// TwinCAT 3 PLC project TcOtel_Tester
// ProgramVersion: 3.1.4026.22
// CompilerDefines: DEBUG
// libraries:
//   TcOtel, * (AVM Engineering)
//   Tc2_Standard, * (Beckhoff Automation GmbH)
//   Tc2_System, * (Beckhoff Automation GmbH)
//   Tc2_Utilities, * (Beckhoff Automation GmbH)
//   Tc3_Module, * (Beckhoff Automation GmbH)
//   Base Interfaces,newest,System
// project tree:
//   GVLs/ GVL.TcGVL, GVL_TracePropagation.TcGVL
//   / PlcTask.TcTTO
//   POUs/ CheckBounds.TcPOU, CheckLRangeSigned.TcPOU, CheckLRangeUnsigned.TcPOU, CheckPointer.TcPOU, CheckRangeSigned.TcPOU, CheckRangeUnsigned.TcPOU, FB_Motor.TcPOU (not stored), FB_TcExternalTime.TcPOU, F_FUN.TcPOU (excluded from build), MAIN.TcPOU (not stored), PRG_TestMetricApi.TcPOU, PRG_TestSimpleApi.TcPOU (not stored), PRG_TestTraceApi.TcPOU, PRG_TestTracePropagation.TcPOU, PRG_TestTracerInstance.TcPOU
// (motion and I/O tree: see PLC project tcotel)
// real-time tasks:
//   TASK PlcTask: cycle T#1ms, priority 20, ADS port 350

CONFIGURATION TcOtel_Tester
    RESOURCE PLC ON TwinCAT3
        TASK PlcTask(INTERVAL := T#1ms, PRIORITY := 20);
        PROGRAM MAIN WITH PlcTask : MAIN;
    END_RESOURCE
END_CONFIGURATION

// ---- GVLs/GVL.TcGVL
{attribute 'qualified_only'}
VAR_GLOBAL
END_VAR

// ---- GVLs/GVL_TracePropagation.TcGVL
(*
Shared state for the Phase-5 cross-task propagation live test
(PRG_TestTracePropagation). Kept in a GVL so one PRG can produce a
traceparent string and another — or a later scenario in the same PRG
— can consume it across cycles.
*)
{attribute 'qualified_only'}
VAR_GLOBAL
    (* Pattern A: explicit W3C traceparent handed off between producer
       and consumer. 55 chars is enough for 00-<32hex>-<16hex>-01. *)
    sCurrentTraceParent : STRING(60);

    (* Pattern D: workpiece-centric trace_id derived via hash of the
       physical workpiece identifier. Modules that can see the ID but
       not a data bus can still aggregate their spans under one
       trace_id. *)
    sWorkpieceId        : STRING(40);
END_VAR

// ---- POUs/PRG_TestTracePropagation.TcPOU
(*
:Description: Phase-5 live cross-task propagation scenarios.

Runs three scenarios on a round-robin cadence so tc-otel sees all
three patterns documented in docs/traces-propagation.md:

  Scenario 1 (Pattern A — explicit traceparent handoff):
    Producer opens a Client span 'order_submit', reads its own
    TraceParent property before End, parks the string in the GVL.
    Consumer later opens 'handle_order' via the FB_Span.Begin
    overload with sTraceParent := the parked string. Tempo should
    render a two-span tree (Client → Server).

  Scenario 2 (Pattern D — workpiece-centric hash):
    Synthesises a workpiece_id like "WP-1234", builds a W3C header
    via F_TraceParentFromString (all-zero span_id — no upstream
    station cited). Opens three module spans across three cycles,
    each passing the same header. Tempo should show one trace with
    three sibling spans sharing a trace_id.

  Scenario 3 (chained producer-consumer-consumer):
    Each stage reads its own TraceParent property before End(),
    passes it to the next stage's Begin. Uses per-instance access
    so parallel Scenarios 1 and 2 on the same task can't poison
    the task-global CurrentTraceParent stack. Tempo shows a linear
    chain A → B → C.

All scenarios use FB_Span methods only — no low-level tracer access.
*)
PROGRAM PRG_TestTracePropagation
VAR
    tracer         : FB_Trace;

    (* Scenario 1: explicit handoff *)
    spnProducer    : FB_Span(tracer);
    spnConsumer    : FB_Span(tracer);
    tScenario1Acc  : TIME;
    nScenario1Step : USINT;  (* 0 idle, 1 producer open, 2 producer ended, 3 consumer open *)

    (* Scenario 2: hash-based, no handoff *)
    spnStageA      : FB_Span(tracer);
    spnStageB      : FB_Span(tracer);
    spnStageC      : FB_Span(tracer);
    tScenario2Acc  : TIME;
    nScenario2Step : USINT;  (* 0..3 *)
    nWorkpieceSeq  : DINT;
    sTraceParentHash : STRING(60);

    (* Scenario 3: chained *)
    spnChainA      : FB_Span(tracer);
    spnChainB      : FB_Span(tracer);
    spnChainC      : FB_Span(tracer);
    tScenario3Acc  : TIME;
    nScenario3Step : USINT;
    sChainTp1      : STRING(60);
    sChainTp2      : STRING(60);

    nSeq           : DINT;
END_VAR


// ─── Scenario 1: explicit traceparent handoff (every 3 s) ───
tScenario1Acc := tScenario1Acc + T#1MS;

CASE nScenario1Step OF
0:  // idle — wait for 3 s cycle start
    IF tScenario1Acc >= T#3S THEN
        tScenario1Acc := T#0S;
        spnProducer.Begin('order_submit', eKind := E_SpanKind.eClient);
        spnProducer.AddInt('seq', nSeq);
        nScenario1Step := 1;
    END_IF
1:  // producer open for ~100 ms, then capture traceparent + end
    IF tScenario1Acc >= T#100MS THEN
        GVL_TracePropagation.sCurrentTraceParent := spnProducer.TraceParent;
        spnProducer.AddEvent('traceparent_captured');
        spnProducer.End();
        nScenario1Step := 2;
    END_IF
2:  // 50 ms gap between producer End and consumer Begin — exercises
    // the "producer already flushed, consumer still opens as child"
    // code path in tc-otel.
    IF tScenario1Acc >= T#150MS THEN
        spnConsumer.Begin(
            sName        := 'handle_order',
            eKind        := E_SpanKind.eServer,
            sTraceParent := GVL_TracePropagation.sCurrentTraceParent);
        spnConsumer.AddInt('seq', nSeq);
		F_Log(E_LogLevel.eDebug, 'Try add trace reference to log entry').WithSpan(spnConsumer).CreateLog();
        nScenario1Step := 3;
    END_IF
3:  // consumer open for ~80 ms, then end + reset
    IF tScenario1Acc >= T#230MS THEN
        spnConsumer.End();
        nSeq := nSeq + 1;
        nScenario1Step := 0;
    END_IF
END_CASE

// ─── Scenario 2: workpiece-centric hash (every 5 s) ───
tScenario2Acc := tScenario2Acc + T#1MS;

CASE nScenario2Step OF
0:
    IF tScenario2Acc >= T#5S THEN
        tScenario2Acc := T#0S;
        GVL_TracePropagation.sWorkpieceId := CONCAT('WP-', DINT_TO_STRING(nWorkpieceSeq));
        nWorkpieceSeq := nWorkpieceSeq + 1;
        // Pattern D helper: hash the workpiece ID into a trace_id, no
        // upstream span to cite (sParentId omitted → all-zero span_id).
        // For a parent-child chain, both producer and consumer must
        // build their traceparent via F_TraceParentFromString with the
        // same sParentId — see docs/traces-propagation.md.
        sTraceParentHash := tc_otel.F_TraceParentFromString(
            sTraceId := GVL_TracePropagation.sWorkpieceId);
        spnStageA.Begin(sName := 'station_weigh', eKind := E_SpanKind.eInternal, sTraceParent := sTraceParentHash);
        spnStageA.AddString('workpiece_id', GVL_TracePropagation.sWorkpieceId);
        nScenario2Step := 1;
    END_IF
1:
    IF tScenario2Acc >= T#50MS THEN
        spnStageA.End();
        spnStageB.Begin(sName := 'station_inspect', eKind := E_SpanKind.eInternal, sTraceParent := sTraceParentHash);
        spnStageB.AddString('workpiece_id', GVL_TracePropagation.sWorkpieceId);
        nScenario2Step := 2;
    END_IF
2:
    IF tScenario2Acc >= T#100MS THEN
        spnStageB.End();
        spnStageC.Begin(sName := 'station_label', eKind := E_SpanKind.eInternal, sTraceParent := sTraceParentHash);
        spnStageC.AddString('workpiece_id', GVL_TracePropagation.sWorkpieceId);
        nScenario2Step := 3;
    END_IF
3:
    IF tScenario2Acc >= T#150MS THEN
        spnStageC.End();
        nScenario2Step := 0;
    END_IF
END_CASE

// ─── Scenario 3: chained producer → consumer → consumer (every 7 s) ───
tScenario3Acc := tScenario3Acc + T#1MS;

CASE nScenario3Step OF
0:
    IF tScenario3Acc >= T#7S THEN
        tScenario3Acc := T#0S;
        spnChainA.Begin('chain_A');
        nScenario3Step := 1;
    END_IF
1:
    IF tScenario3Acc >= T#60MS THEN
        sChainTp1 := spnChainA.TraceParent;
        spnChainA.End();
        spnChainB.Begin(sName := 'chain_B', sTraceParent := sChainTp1);
        nScenario3Step := 2;
    END_IF
2:
    IF tScenario3Acc >= T#120MS THEN
        sChainTp2 := spnChainB.TraceParent;
        spnChainB.End();
        spnChainC.Begin(sName := 'chain_C', sTraceParent := sChainTp2);
        nScenario3Step := 3;
    END_IF
3:
    IF tScenario3Acc >= T#180MS THEN
        spnChainC.End();
        nScenario3Step := 0;
    END_IF
END_CASE

END_PROGRAM

// ---- POUs/CheckBounds.TcPOU
// Implicitly generated code : DO NOT EDIT
FUNCTION CheckBounds : DINT
VAR_INPUT
	index, lower, upper: DINT;
END_VAR

{noflow}
IF (index < lower) THEN
	CheckBounds := lower;
	F_Log(E_LogLevel.eFatal, 'Check bounds exception: {index} {lower} {upper}').WithLogger('CheckBounds').WithAnyArg(index).WithAnyArg(lower).WithAnyArg(upper).CreateLog();
ELSIF(index > upper) THEN
	CheckBounds := upper;
	F_Log(E_LogLevel.eFatal, 'Check bounds exception: {index} {lower} {upper}').WithLogger('CheckBounds').WithAnyArg(index).WithAnyArg(lower).WithAnyArg(upper).CreateLog();
ELSE
	CheckBounds := index;
END_IF
{flow}

END_FUNCTION

// ---- POUs/CheckLRangeSigned.TcPOU
// Implicitly generated code : DO NOT EDIT
FUNCTION CheckLRangeSigned : LINT
VAR_INPUT
	value, lower, upper: LINT;
END_VAR

{noflow}
IF (value < lower) THEN
	CheckLRangeSigned := lower;
	F_Log(E_LogLevel.eFatal, 'Check LINT range signed exception: {value} {lower} {upper}').WithLogger('CheckLRangeSigned').WithAnyArg(value).WithAnyArg(lower).WithAnyArg(upper).CreateLog();
ELSIF(value > upper) THEN
	CheckLRangeSigned := upper;
	F_Log(E_LogLevel.eFatal, 'Check LINT range signed exception: {value} {lower} {upper}').WithLogger('CheckLRangeSigned').WithAnyArg(value).WithAnyArg(lower).WithAnyArg(upper).CreateLog();
ELSE
	CheckLRangeSigned := value;
END_IF
{flow}

END_FUNCTION

// ---- POUs/CheckLRangeUnsigned.TcPOU
// Implicitly generated code : DO NOT EDIT
FUNCTION CheckLRangeUnsigned : ULINT
VAR_INPUT
	value, lower, upper: ULINT;
END_VAR

{noflow}
IF (value < lower) THEN
	CheckLRangeUnsigned := lower;
	F_Log(E_LogLevel.eFatal, 'Check ULINT range unsigned exception: {value} {lower} {upper}').WithLogger('CheckLRangeUnsigned').WithAnyArg(value).WithAnyArg(lower).WithAnyArg(upper).CreateLog();
ELSIF(value > upper) THEN
	CheckLRangeUnsigned := upper;
	F_Log(E_LogLevel.eFatal, 'Check ULINT range unsigned exception: {value} {lower} {upper}').WithLogger('CheckLRangeUnsigned').WithAnyArg(value).WithAnyArg(lower).WithAnyArg(upper).CreateLog();
ELSE
	CheckLRangeUnsigned := value;
END_IF
{flow}

END_FUNCTION

// ---- POUs/CheckPointer.TcPOU
// Implicitly generated code : DO NOT EDIT
FUNCTION CheckPointer : POINTER TO BYTE
VAR_INPUT 
	ptToTest : POINTER TO BYTE; // Destination address of the pointer
	iSize : DINT;		        // Size of the type the pointer points to. (e.g: 20 for POINTER TO ARRAY [0..9] OF INT) 
	iGran : DINT;		        // Granularity of the pointer access. This is the size of the biggest non-structured data type in the type the pointer points to. (e.g: 2 for POINTER TO ARRAY [0..9] OF INT)
	bWrite: BOOL;		        // Indicates read or write Access. TRUE = write access.
END_VAR

IF ptToTest = 0 THEN
	F_Log(E_LogLevel.eFatal, 'Check pointer exception: {iSize} {iGran} {bWrite}').WithLogger('CheckPointer').WithAnyArg(iSize).WithAnyArg(iGran).WithAnyArg(bWrite).CreateLog();
END_IF
CheckPointer := ptToTest;

END_FUNCTION

// ---- POUs/CheckRangeSigned.TcPOU
// Implicitly generated code : DO NOT EDIT
FUNCTION CheckRangeSigned : DINT
VAR_INPUT
	value, lower, upper: DINT;
END_VAR

{noflow}
IF (value < lower) THEN
	CheckRangeSigned := lower;
	F_Log(E_LogLevel.eFatal, 'Check DINT range signed exception: {value} {lower} {upper}').WithLogger('CheckRangeSigned').WithAnyArg(value).WithAnyArg(lower).WithAnyArg(upper).CreateLog();
ELSIF(value > upper) THEN
	CheckRangeSigned := upper;
	F_Log(E_LogLevel.eFatal, 'Check DINT range signed exception: {value} {lower} {upper}').WithLogger('CheckRangeSigned').WithAnyArg(value).WithAnyArg(lower).WithAnyArg(upper).CreateLog();
ELSE
	CheckRangeSigned := value;
END_IF
{flow}

END_FUNCTION

// ---- POUs/CheckRangeUnsigned.TcPOU
// Implicitly generated code : DO NOT EDIT
FUNCTION CheckRangeUnsigned : UDINT
VAR_INPUT
	value, lower, upper: UDINT;
END_VAR

{noflow}
IF (value < lower) THEN
	CheckRangeUnsigned := lower;
	F_Log(E_LogLevel.eFatal, 'Check UDINT range unsigned exception: {value} {lower} {upper}').WithLogger('CheckRangeUnsigned').WithAnyArg(value).WithAnyArg(lower).WithAnyArg(upper).CreateLog();
ELSIF(value > upper) THEN
	CheckRangeUnsigned := upper;
	F_Log(E_LogLevel.eFatal, 'Check UDINT range unsigned exception: {value} {lower} {upper}').WithLogger('CheckRangeUnsigned').WithAnyArg(value).WithAnyArg(lower).WithAnyArg(upper).CreateLog();
ELSE
	CheckRangeUnsigned := value;
END_IF
{flow}

END_FUNCTION

// ---- POUs/FB_TcExternalTime.TcPOU
FUNCTION_BLOCK FB_TcExternalTime
VAR
	_hr : HRESULT;
	_ipExtTime : ITcExternalTime;
	_eTimeType: ETcExternalTimeType;
END_VAR

METHOD FB_Exit : BOOL
VAR_INPUT
	bInCopyCode : BOOL; // if TRUE, the exit method is called for exiting an instance that is copied afterwards (online change).
END_VAR
IF _ipExtTime <> 0 THEN
	FW_SafeRelease(ADR(_ipExtTime));
END_IF
END_METHOD

METHOD FB_Init : BOOL
VAR_INPUT
	bInitRetains : BOOL; // if TRUE, the retain variables are initialized (warm start / cold start)
	bInCopyCode : BOOL;  // if TRUE, the instance afterwards gets moved into the copy code (online change)
	eTimeType : ETcExternalTimeType; 
END_VAR
VAR
	ipServer : ITComObjectServer;
END_VAR
ipServer := TwinCAT_SystemInfoVarList._AppInfo.TComSrvPtr;
_eTimeType := eTimeType; 
IF _ipExtTime = 0 THEN
	_hr := ipServer.TcQueryInterface(IID_ITcExternalTime, ADR(_ipExtTime));
	IF FAILED(_hr) THEN RETURN; END_IF
END_IF
END_METHOD

METHOD GetExternalOffset : LINT
VAR_INPUT
END_VAR
IF _ipExtTime <> 0 THEN
	_hr := _ipExtTime.GetExternalTimeOffset(_eTimeType, GetExternalOffset);
	IF _hr <> 0 THEN GetExternalOffset := 0; END_IF
END_IF
END_METHOD

METHOD GetExternalTime : LINT
VAR_INPUT
END_VAR
IF _ipExtTime <> 0 THEN
	GetExternalTime := GetSystemTime();
	_hr := _ipExtTime.SystemTimeToExternalTime(_eTimeType, GetExternalTime);
	IF _hr <> 0 THEN GetExternalTime := 0; END_IF
END_IF
END_METHOD

METHOD GetSystemTime : LINT
GetSystemTime := ULINT_TO_LINT(F_GetSystemTime());
END_METHOD

PROPERTY Result : HRESULT
GET
Result := _hr;
END_GET
END_PROPERTY

END_FUNCTION_BLOCK

// ---- POUs/F_FUN.TcPOU
FUNCTION F_FUN : BOOL
VAR_INPUT
END_VAR
VAR
	var1			: __SYSTEM.VAR_INFO;
	var2			: __SYSTEM.VAR_INFO;
	fbLog			: FB_Logger('F_FUN (Inst)');
END_VAR
VAR_STAT
	fbLog2			: FB_Logger('F_FUN (Stat)');
END_VAR

fbLog();
fbLog2();
var1 := __VARINFO(fbLog);
var2 := __VARINFO(fbLog2);

END_FUNCTION

// ---- POUs/PRG_TestMetricApi.TcPOU
PROGRAM PRG_TestMetricApi
VAR
	(* FB_Metrics smoke instances — exercise each body schema. *)
	fbSineLreal     : FB_Metrics;
	fbToggleBool    : FB_Metrics;
	fbStateString   : FB_Metrics;
	(* Phase 7: same sine fed into an aggregating instance — the receiver
	   sees min/max/mean per sample tick instead of an under-sampled raw
	   value, so the envelope stays sharp even at 50 ms / 5 s cadence. *)
	fbSineAgg       : FB_Metrics;

	(* Driver state. *)
	rPhase          : LREAL;
	rSineValue      : LREAL;
	bToggle         : BOOL;
	sState          : STRING(31) := 'idle';
	nStateSwitch    : UDINT;
END_VAR

IF TwinCAT_SystemInfoVarList._TaskInfo[GETCURTASKINDEXEX()].FirstCycle THEN
	// FB_Metrics demo: LREAL sine → eNumeric body schema, push every 5 s.
	fbSineLreal.Init('demo.sine', 'unit');
	fbSineLreal.SetSampleIntervalMs(50);
	fbSineLreal.SetPushIntervalMs(5000);

	// BOOL toggle → eBool, push every 2 s.
	fbToggleBool.Init('demo.toggle', '');
	fbToggleBool.SetPushIntervalMs(2000);

	// STRING state → eString (fixed 32 B per sample), push every 10 s.
	fbStateString.Init('demo.state', '', 32);
	fbStateString.SetPushIntervalMs(10000);

	// Aggregated sine: same source, same 50 ms / 5 s cadence — but
	// SetAggregation(eMin OR eMax OR eMean) folds every Observe into
	// Welford online so each sample tick captures the real envelope of
	// the underlying signal instead of a stochastic point on it.
	fbSineAgg.Init('demo.sineAgg', 'unit');
	fbSineAgg.SetSampleIntervalMs(50);
	fbSineAgg.SetPushIntervalMs(5000);
	fbSineAgg.SetAggregation(E_MetricStat.eMean OR E_MetricStat.eMax OR E_MetricStat.eMin);
END_IF

// Drive the sine: phase advances 0.005 rad per 1 ms task cycle ≈ 0.8 Hz.
// Combined with SetSampleIntervalMs(50) → ~25 samples per period — clean
// curve in Grafana (well above Nyquist, no visible aliasing).
rPhase     := rPhase + 0.005;
rSineValue := SIN(rPhase);
fbSineLreal.Observe(rSineValue);
fbSineAgg.Observe(rSineValue);

// BOOL toggles every 250 cycles for an obvious square wave on the wire.
IF (TwinCAT_SystemInfoVarList._TaskInfo[GETCURTASKINDEXEX()].CycleCount MOD 250) = 0 THEN
	bToggle := NOT bToggle;
END_IF
fbToggleBool.Observe(bToggle);

// State machine flips through 3 strings every ~3 s (3000 cycles at 1 ms).
nStateSwitch := nStateSwitch + 1;
IF nStateSwitch >= 3000 THEN
	nStateSwitch := 0;
	IF sState = 'idle' THEN
		sState := 'running';
	ELSIF sState = 'running' THEN
		sState := 'paused';
	ELSE
		sState := 'idle';
	END_IF
END_IF
fbStateString.Observe(sState);

END_PROGRAM

// ---- POUs/PRG_TestTraceApi.TcPOU
PROGRAM PRG_TestTraceApi
VAR
    tracer        : FB_Trace;
    spnTick       : FB_Span(tracer);
    spnRecipe     : FB_Span(tracer);
    spnRecipeStep : FB_Span(tracer);
    tTickAccum    : TIME;
    tRecipeAccum  : TIME;
    nSeq          : DINT;
    nRecipeStep   : DINT;
    bRecipeActive : BOOL;
END_VAR


// --- 1 Hz tick span: demonstrates a simple single-cycle span every second ---
tTickAccum := tTickAccum + T#1MS;
IF tTickAccum >= T#1S THEN
    tTickAccum := T#0S;
    spnTick.Begin('tester_1s_tick');
    spnTick.AddInt('seq', nSeq);
    spnTick.AddEvent('midpoint');
    spnTick.End();
    nSeq := nSeq + 1;
END_IF

// --- 5 s nested-span demo: demonstrates parent/child relationship over multiple cycles ---
tRecipeAccum := tRecipeAccum + T#1MS;
IF NOT bRecipeActive AND tRecipeAccum >= T#5S THEN
    tRecipeAccum := T#0S;
    spnRecipe.Begin('tester_recipe', eKind := E_SpanKind.eInternal);
    spnRecipe.AddString('mode', 'nested_demo');
    bRecipeActive := TRUE;
    nRecipeStep := 0;
END_IF

IF bRecipeActive THEN
    // One nested step per second for 3 seconds, then end the outer recipe
    IF spnRecipeStep.IsOpen THEN
        // Inner span runs for ~300 ms from its Begin
        IF TIME_TO_UDINT(tRecipeAccum) MOD 1000 >= 300 THEN
            spnRecipeStep.AddEvent('inner_done');
            spnRecipeStep.End();
        END_IF
    ELSE
        IF nRecipeStep < 3 AND TIME_TO_UDINT(tRecipeAccum) MOD 1000 = 0 THEN
            spnRecipeStep.Begin(CONCAT('step_', DINT_TO_STRING(nRecipeStep)));
            spnRecipeStep.AddInt('step_idx', nRecipeStep);
            nRecipeStep := nRecipeStep + 1;
        END_IF
    END_IF

    IF nRecipeStep >= 3 AND NOT spnRecipeStep.IsOpen THEN
        spnRecipe.AddEvent('all_steps_done');
        spnRecipe.End();
        bRecipeActive := FALSE;
    END_IF
END_IF

END_PROGRAM

// ---- POUs/PRG_TestTracerInstance.TcPOU
(*
:Description: Phase 6 Stage 1 live verification — two parallel
FB_TcOtelTracer instances on the same task, each running their own
nested span chain.

Before Stage 1, this scenario would have been impossible: both
controllers' spans would push onto the task-global aStack and
either contaminate each other's CurrentTraceParent or use each
other as parent in nested Begin calls. With BindTracer, each
controller's span tree is isolated.

Expectation in Tempo:
* Two separate traces (distinct trace_ids) every cycle.
* Controller A: ``ctl_a_outer`` with nested ``ctl_a_inner``.
* Controller B: ``ctl_b_outer`` with nested ``ctl_b_inner``.
* ``ctl_a_inner`` parent = ``ctl_a_outer`` (never ctl_b_outer).
* ``ctl_b_inner`` parent = ``ctl_b_outer`` (never ctl_a_outer).
*)
PROGRAM PRG_TestTracerInstance
VAR
    tAccum        : TIME;
    nStep         : USINT;

    (* Controller A: tracer + its two spans *)
    tracerA       : FB_Trace;
    spnAOuter     : FB_Span(tracerA);
    spnAInner     : FB_Span(tracerA);

    (* Controller B: tracer + its two spans *)
    tracerB       : FB_Trace;
    spnBOuter     : FB_Span(tracerB);
    spnBInner     : FB_Span(tracerB);
END_VAR

tAccum := tAccum + T#1MS;

// Every 4 s run the interleaved dance. Both controllers open outer,
// open inner, close inner, close outer — but in shuffled order so
// any stack-based parent resolution would pair them wrong.
CASE nStep OF
0:
    IF tAccum >= T#4S THEN
        tAccum := T#0S;
        spnAOuter.Begin('ctl_a_outer');
        nStep := 1;
    END_IF
1:
    IF tAccum >= T#20MS THEN
        // B opens BEFORE A has opened its inner. If FB_Span used
        // the task-global stack, spnAInner (below) would inherit
        // from spnBOuter. With per-tracer nesting it won't.
        spnBOuter.Begin('ctl_b_outer');
        nStep := 2;
    END_IF
2:
    IF tAccum >= T#40MS THEN
        // A's inner must see spnAOuter as parent, not spnBOuter.
        spnAInner.Begin('ctl_a_inner');
        nStep := 3;
    END_IF
3:
    IF tAccum >= T#60MS THEN
        // B's inner must see spnBOuter as parent.
        spnBInner.Begin('ctl_b_inner');
        nStep := 4;
    END_IF
4:
    IF tAccum >= T#80MS THEN
        spnAInner.End();    // close inner-A first
        nStep := 5;
    END_IF
5:
    IF tAccum >= T#100MS THEN
        spnBInner.End();    // close inner-B
        nStep := 6;
    END_IF
6:
    IF tAccum >= T#120MS THEN
        spnBOuter.End();    // close outer-B out of order
        nStep := 7;
    END_IF
7:
    IF tAccum >= T#140MS THEN
        spnAOuter.End();    // close outer-A last
        nStep := 0;
    END_IF
END_CASE

END_PROGRAM
